(* IEC 61131-3 sources: CodesysTest/export/ObjectHandling/FB_CollectionHandlerFaults.pou, 3 files *)

(* ---- FB_CollectionHandlerFaults.pou.st ---- *)
(*#-#-#-#-#-#-#-#-#-#---Declaration---#-#-#-#-#-#-#-#-#-#-#-#-#*)

FUNCTION_BLOCK FB_CollectionHandlerFaults
VAR_INPUT
END_VAR
VAR
	Collection: ARRAY[0..GlobalObjects.MAX_FAULTS] OF IFault; // object array
	ObjNames   : ARRAY[0..GlobalObjects.MAX_FAULTS] OF STRING;
	faults : ARRAY[0..GlobalObjects.MAX_FAULTS] OF HMIFaultType;
	_ArrayOver   : BOOL;
	_BadObj      : INT;
	_DupeObj   : INT;
	_OverObj   : INT;
	_TotalObj   : UINT;
	_InitFaultList : BOOL;
END_VAR(*#-#-#-#-#-#-#-#-#-#---Implementation---#-#-#-#-#-#-#-#-#-#-#-#-#*)

(* ---- AckAll.m.st ---- *)
(*#-#-#-#-#-#-#-#-#-#---Declaration---#-#-#-#-#-#-#-#-#-#-#-#-#*)

METHOD AckAll
VAR_INPUT
END_VAR
VAR
	Cast : IFault;
	Fault : IFault;
	J : UINT;
END_VAR(*#-#-#-#-#-#-#-#-#-#---Implementation---#-#-#-#-#-#-#-#-#-#-#-#-#*)

// For each active fault in the array, ack it.
IF _TotalObj <=0 THEN
	RETURN;
END_IF
FOR J:= 0 TO _TotalObj - 1 DO
		Collection[J].Ack();
END_FOR

(* ---- FaultUpdateForHMI.m.st ---- *)
(*#-#-#-#-#-#-#-#-#-#---Declaration---#-#-#-#-#-#-#-#-#-#-#-#-#*)

METHOD FaultUpdateForHMI
VAR_INPUT
END_VAR
VAR
	I : UINT;
END_VAR(*#-#-#-#-#-#-#-#-#-#---Implementation---#-#-#-#-#-#-#-#-#-#-#-#-#*)

FOR I:= 0 TO _TotalObj - 1 DO
	IF NOT _InitFaultList THEN
		faults[I].name := Collection[I].InstanceName;
	END_IF
	faults[I].active := Collection[I].FaultActive;
END_FOR
_InitFaultList := TRUE;
